// TIA Portal V20 export
TYPE "type_emRelations_em7_cmStatus"
// stored: Access Published, Namespace Unit1
   STRUCT
      HotPressRightSafetyPin : "LBC_typeDigitalSignalControlNode";
      HotPressRightJRDetect : "LBC_typeDigitalSignalControlNode";
      HotPressRightStageLiftFrontUpDown : "LBC_typeTwoWayActuatorControlNode";
      HotPressRightStageLiftRearUpDown : "LBC_typeTwoWayActuatorControlNode";
      HotPressRightStageLiftAllUpDown : "LBC_typeTwoWayActuatorControlNode";
      HotPressRightServoPress : "LER_typeServoPressControlNode";
      HotPressRightTemperature : "LER_typeHeaterControlNode";
   END_STRUCT;
END_TYPE
